    rq_wait_ft_sensor_steady(2000)
    zero_ftsensor()
    sleep(0.1)
    # end: URCap Program Node
    # begin: URCap Program Node
    #   Source: Robotiq_Copilot, 1.22.1.14215, Robotiq Inc.
    #   Type: Find Surface
    $ 80 "Find Surface"
    zero_ftsensor()
    sleep(0.1)
    surface_found = rq_linear_search_urcap("Z+", 10.000, 0.005000, 0.100000, 1)
    storevar.setvariablepose("rq_findSurface_ef5e6fd5-1d3d-43c2-9922-b9c2fd55821a_exitPosition", get_actual_tcp_pose())
    $ 81 "'Add Stop conditions from the Find Surface node'" "noBreak"
    # 'Add Stop conditions from the Find Surface node'
    # end: URCap Program Node
    # begin: URCap Program Node
    #   Source: Robotiq_Copilot, 1.22.1.14215, Robotiq Inc.
    #   Type: Finishing Tool Control
    $ 82 "Start tool"
    set_standard_digital_out(0, True)
    # end: URCap Program Node
    $ 83 "Wait: 0.5"
    sleep(0.5)
    $ 84 "Force"
    sleep(0.02)
    zero_ftsensor()
    force_mode(tool_pose(), [0, 0, 1, 0, 0, 0], [0.0, 0.0, 5.0, 0.0, 0.0, 0.0], 2, [0.1, 0.1, 0.15, 0.3490658503988659, 0.3490658503988659, 0.3490658503988659])
    $ 85 "Waypoint_7" "noBreak"
    set_tcp(p[0.00318,0.11464,0.09820000000000001,-0.7853981633974483,0.0,0.0])
    movel(pose_trans(CubeFront, pose_trans(p[-.005597006121, -.192408094989, .653246871754, -1.571622694982, -.002967386491, .002471774867], Waypoint_7_p)), a=1.2, v=0.05)
    end_force_mode()
    stopl(5.0)
    # begin: URCap Program Node
    #   Source: Robotiq_Copilot, 1.22.1.14215, Robotiq Inc.
    #   Type: Finishing Tool Control
    $ 86 "Stop tool"
    set_standard_digital_out(0, False)
    # end: URCap Program Node
    $ 87 "Waypoint_13" "breakAfter"
    set_tcp(p[0.00318,0.11464,0.09820000000000001,-0.7853981633974483,0.0,0.0])
    movel(pose_trans(CubeFront, pose_trans(p[-.002001169423, -.178123008725, .618090231485, -1.568699287997, .013964727372, .007428573496], Waypoint_13_p)), a=1.2, v=0.25)
    $ 88 "Waypoint_9" "breakAfter"
    set_tcp(p[0.00318,0.11464,0.09820000000000001,-0.7853981633974483,0.0,0.0])
    movel(pose_trans(CubeFront, pose_trans(p[-.002001169423, -.178123008725, .618090231485, -1.568699287997, .013964727372, .007428573496], Waypoint_9_p)), a=1.2, v=0.25)
    $ 89 "clear" "breakAfter"
    set_tcp(p[0.00318,0.11464,0.09820000000000001,-0.7853981633974483,0.0,0.0])
    movel(pose_trans(CubeFront, pose_trans(p[.002249871974, -.169402369556, .608081756259, .020435046430, 2.223511403835, 2.209446612627], clear_p)), a=1.2, v=0.25)
  end
  def SprayFront():
    $ 90 "SprayFront" "noBreak"
    $ 91 "SprayFront"
    $ 92 "MoveJ"
    $ 93 "clear" "breakAfter"
    set_tcp(p[0.00318,0.11464,0.09820000000000001,-0.7853981633974483,0.0,0.0])
    movej(get_inverse_kin(pose_trans(CubeFront, pose_trans(p[.002249871974, -.169402369556, .608081756259, .020435046430, 2.223511403835, 2.209446612627], clear_p)), qnear=clear_q), a=1.3962634015954636, v=1.0471975511965976)
    $ 94 "MoveJ"
    $ 95 "Waypoint_10" "breakAfter"
    set_tcp(p[0.020839023181949995,-0.027139950822234082,0.10599373590389219,0.12258870209179472,1.1769383890382668,2.869747076630172])
    movej(get_inverse_kin(pose_trans(CubeFront, pose_trans(p[-.002001169423, -.178123008725, .618090231485, -1.568699287997, .013964727372, .007428573496], Waypoint_10_p)), qnear=Waypoint_10_q), a=1.3962634015954636, v=1.0471975511965976)
    $ 96 "Set DO[1]=On"
    set_standard_digital_out(1, True)
    $ 97 "MoveL"
    $ 98 "Waypoint_12" "breakAfter"
    movel(pose_trans(CubeFront, pose_trans(p[-.002001169423, -.178123008725, .618090231485, -1.568699287997, .013964727372, .007428573496], Waypoint_12_p)), a=1.2, v=0.1)
    $ 99 "Set DO[1]=Off"
    set_standard_digital_out(1, False)
    $ 100 "MoveJ"
    $ 101 "Waypoint_21" "breakAfter"
    set_tcp(p[0.020839023181949995,-0.027139950822234082,0.10599373590389219,0.12258870209179472,1.1769383890382668,2.869747076630172])
    movej(get_inverse_kin(pose_trans(CubeFront, pose_trans(p[-.002001169423, -.178123008725, .618090231485, -1.568699287997, .013964727372, .007428573496], Waypoint_21_p)), qnear=Waypoint_21_q), a=1.3962634015954636, v=1.0471975511965976)
    $ 102 "Set DO[1]=On"
    set_standard_digital_out(1, True)
    $ 103 "MoveL"
    $ 104 "Waypoint_22" "breakAfter"
    set_tcp(p[0.020839023181949995,-0.027139950822234082,0.10599373590389219,0.12258870209179472,1.1769383890382668,2.869747076630172])
    movel(pose_trans(CubeFront, pose_trans(p[-.002001169423, -.178123008725, .618090231485, -1.568699287997, .013964727372, .007428573496], Waypoint_22_p)), a=1.2, v=0.1)
    $ 105 "Set DO[1]=Off"
    set_standard_digital_out(1, False)
    $ 106 "MoveJ"
    $ 107 "Waypoint_23" "breakAfter"
    set_tcp(p[0.020839023181949995,-0.027139950822234082,0.10599373590389219,0.12258870209179472,1.1769383890382668,2.869747076630172])
    movej(get_inverse_kin(pose_trans(CubeFront, pose_trans(p[-.002001169423, -.178123008725, .618090231485, -1.568699287997, .013964727372, .007428573496], Waypoint_23_p)), qnear=Waypoint_23_q), a=1.3962634015954636, v=1.0471975511965976)
    $ 108 "Set DO[1]=On"
    set_standard_digital_out(1, True)
    $ 109 "MoveL"
    $ 110 "Waypoint_24" "breakAfter"
    set_tcp(p[0.020839023181949995,-0.027139950822234082,0.10599373590389219,0.12258870209179472,1.1769383890382668,2.869747076630172])
    movel(pose_trans(CubeFront, pose_trans(p[-.002001169423, -.178123008725, .618090231485, -1.568699287997, .013964727372, .007428573496], Waypoint_24_p)), a=1.2, v=0.1)
    $ 111 "Set DO[1]=Off"
    set_standard_digital_out(1, False)
    $ 112 "MoveJ"
    $ 113 "clear" "breakAfter"
    movej(clear_q, a=1.3962634015954636, v=1.0471975511965976)
    $ 114 "MoveJ"
    $ 115 "Waypoint_26" "breakAfter"
    set_tcp(p[0.020839023181949995,-0.027139950822234082,0.10599373590389219,0.12258870209179472,1.1769383890382668,2.869747076630172])
    movej(get_inverse_kin(pose_trans(CubeFront, pose_trans(p[-.002001169423, -.178123008725, .618090231485, -1.568699287997, .013964727372, .007428573496], Waypoint_26_p)), qnear=Waypoint_26_q), a=1.3962634015954636, v=1.0471975511965976)
    $ 116 "Set DO[1]=On"
    set_standard_digital_out(1, True)
    $ 117 "MoveL"
    $ 118 "Waypoint_25" "breakAfter"
    set_tcp(p[0.020839023181949995,-0.027139950822234082,0.10599373590389219,0.12258870209179472,1.1769383890382668,2.869747076630172])
    movel(pose_trans(CubeFront, pose_trans(p[-.002001169423, -.178123008725, .618090231485, -1.568699287997, .013964727372, .007428573496], Waypoint_25_p)), a=1.2, v=0.1)
    $ 119 "Set DO[1]=Off"
    set_standard_digital_out(1, False)
    $ 120 "MoveJ"
    $ 121 "clear" "breakAfter"
    movej(clear_q, a=1.3962634015954636, v=1.0471975511965976)
  end
  def SprayRebate():
    $ 122 "SprayRebate" "noBreak"
    $ 123 "SprayRebate"
    $ 124 "MoveJ"
    $ 125 "clear" "breakAfter"
    movej(clear_q, a=1.3962634015954636, v=1.0471975511965976)
    $ 126 "MoveJ"
    $ 127 "Waypoint_28" "breakAfter"
    set_tcp(p[0.020839023181949995,-0.027139950822234082,0.10599373590389219,0.12258870209179472,1.1769383890382668,2.869747076630172])
    movej(get_inverse_kin(pose_trans(CubeFront, pose_trans(p[-.002001169423, -.178123008725, .618090231485, -1.568699287997, .013964727372, .007428573496], Waypoint_28_p)), qnear=Waypoint_28_q), a=1.3962634015954636, v=1.0471975511965976)
    $ 128 "Set DO[1]=On"
    set_standard_digital_out(1, True)
    $ 129 "MoveL"
    $ 130 "Waypoint_27" "breakAfter"
    set_tcp(p[0.020839023181949995,-0.027139950822234082,0.10599373590389219,0.12258870209179472,1.1769383890382668,2.869747076630172])
    movel(pose_trans(CubeFront, pose_trans(p[-.002001169423, -.178123008725, .618090231485, -1.568699287997, .013964727372, .007428573496], Waypoint_27_p)), a=1.2, v=0.1)
    $ 131 "Set DO[1]=Off"
    set_standard_digital_out(1, False)
    $ 132 "MoveJ"
    $ 133 "Waypoint_29" "breakAfter"
    set_tcp(p[0.020839023181949995,-0.027139950822234082,0.10599373590389219,0.12258870209179472,1.1769383890382668,2.869747076630172])
    movej(get_inverse_kin(pose_trans(CubeFront, pose_trans(p[-.002001169423, -.178123008725, .618090231485, -1.568699287997, .013964727372, .007428573496], Waypoint_29_p)), qnear=Waypoint_29_q), a=1.3962634015954636, v=1.0471975511965976)
    $ 134 "Set DO[1]=On"
    set_standard_digital_out(1, True)
    $ 135 "MoveL"
    $ 136 "Waypoint_30" "breakAfter"
    set_tcp(p[0.020839023181949995,-0.027139950822234082,0.10599373590389219,0.12258870209179472,1.1769383890382668,2.869747076630172])
    movel(pose_trans(CubeFront, pose_trans(p[-.002001169423, -.178123008725, .618090231485, -1.568699287997, .013964727372, .007428573496], Waypoint_30_p)), a=1.2, v=0.1)
    $ 137 "Set DO[1]=Off"
    set_standard_digital_out(1, False)
    $ 138 "MoveJ"
    $ 139 "clear" "breakAfter"
    movej(clear_q, a=1.3962634015954636, v=1.0471975511965976)
    $ 140 "MoveJ"
    $ 141 "Waypoint_32" "breakAfter"
    set_tcp(p[0.020839023181949995,-0.027139950822234082,0.10599373590389219,0.12258870209179472,1.1769383890382668,2.869747076630172])
    movej(get_inverse_kin(pose_trans(CubeFront, pose_trans(p[-.002001169423, -.178123008725, .618090231485, -1.568699287997, .013964727372, .007428573496], Waypoint_32_p)), qnear=Waypoint_32_q), a=1.3962634015954636, v=1.0471975511965976)
    $ 142 "Set DO[1]=On"
    set_standard_digital_out(1, True)
    $ 143 "MoveL"
    $ 144 "Waypoint_33" "breakAfter"
    set_tcp(p[0.020839023181949995,-0.027139950822234082,0.10599373590389219,0.12258870209179472,1.1769383890382668,2.869747076630172])
    movel(pose_trans(CubeFront, pose_trans(p[-.002001169423, -.178123008725, .618090231485, -1.568699287997, .013964727372, .007428573496], Waypoint_33_p)), a=1.2, v=0.1)
    $ 145 "Set DO[1]=Off"
    set_standard_digital_out(1, False)
    $ 146 "MoveJ"
    $ 147 "clear" "breakAfter"
    movej(clear_q, a=1.3962634015954636, v=1.0471975511965976)
  end
  def SandFront():
    $ 148 "SandFront" "noBreak"
    $ 149 "sandFront"
    $ 150 "MoveJ"
    $ 151 "clear" "breakAfter"
    set_tcp(p[0.00318,0.11464,0.09820000000000001,-0.7853981633974483,0.0,0.0])
    movej(get_inverse_kin(pose_trans(CubeFront, pose_trans(p[.002249871974, -.169402369556, .608081756259, .020435046430, 2.223511403835, 2.209446612627], clear_p)), qnear=clear_q), a=1.3962634015954636, v=1.0471975511965976)
    $ 152 "MoveL"
    $ 153 "Waypoint_1" "breakAfter"
    set_tcp(p[0.00318,0.11464,0.09820000000000001,-0.7853981633974483,0.0,0.0])
    movel(pose_trans(CubeFront, pose_trans(p[-.005597006121, -.192408094989, .653246871754, -1.571622694982, -.002967386491, .002471774867], Waypoint_1_p)), a=1.2, v=0.25)
    # begin: URCap Program Node
    #   Source: Robotiq_Copilot, 1.22.1.14215, Robotiq Inc.
    #   Type: Zero FT Sensor
    $ 154 "Zero FT Sensor"

    rq_wait_ft_sensor_steady(2000)
    zero_ftsensor()
    sleep(0.1)
    # end: URCap Program Node
    # begin: URCap Program Node
    #   Source: Robotiq_Copilot, 1.22.1.14215, Robotiq Inc.
    #   Type: Find Surface
    $ 155 "Find Surface"
    surface_found = rq_linear_search_urcap("Z+", 10.000, 0.005000, 0.100000, 1)
    storevar.setvariablepose("rq_findSurface_7eeff1a3-6c12-4ed4-8857-ddcfb00799c6_exitPosition", get_actual_tcp_pose())
    $ 156 "'Add Stop conditions from the Find Surface node'" "noBreak"
    # 'Add Stop conditions from the Find Surface node'
    # end: URCap Program Node
    # begin: URCap Program Node
    #   Source: Robotiq_Copilot, 1.22.1.14215, Robotiq Inc.
    #   Type: Finishing Tool Control
    $ 157 "Start tool"
    set_standard_digital_out(0, True)
    # end: URCap Program Node
    $ 158 "Wait: 0.5"
    sleep(0.5)
    $ 159 "MoveL"
    $ 160 "Force"
    sleep(0.02)
    zero_ftsensor()
    force_mode(tool_pose(), [0, 0, 1, 0, 0, 0], [0.0, 0.0, 5.0, 0.0, 0.0, 0.0], 2, [0.1, 0.1, 0.15, 0.3490658503988659, 0.3490658503988659, 0.3490658503988659])
    $ 161 "Waypoint_34" "noBreak"
    set_tcp(p[0.00318,0.11464,0.09820000000000001,-0.7853981633974483,0.0,0.0])
    movel(pose_trans(CubeFront, pose_trans(p[.002249871974, -.169402369556, .608081756259, .020435046430, 2.223511403835, 2.209446612627], Waypoint_34_p)), a=1.2, v=0.06)
    $ 162 "Waypoint_37" "noBreak"
    set_tcp(p[0.00318,0.11464,0.09820000000000001,-0.7853981633974483,0.0,0.0])
    movel(pose_trans(CubeFront, pose_trans(p[.002249871974, -.169402369556, .608081756259, .020435046430, 2.223511403835, 2.209446612627], Waypoint_37_p)), a=1.2, v=0.06)
    $ 163 "Waypoint_36" "noBreak"
    set_tcp(p[0.00318,0.11464,0.09820000000000001,-0.7853981633974483,0.0,0.0])
    movel(pose_trans(CubeFront, pose_trans(p[.002249871974, -.169402369556, .608081756259, .020435046430, 2.223511403835, 2.209446612627], Waypoint_36_p)), a=1.2, v=0.06)
    $ 164 "Waypoint_1" "noBreak"
    set_tcp(p[0.00318,0.11464,0.09820000000000001,-0.7853981633974483,0.0,0.0])
    movel(pose_trans(CubeFront, pose_trans(p[-.005597006121, -.192408094989, .653246871754, -1.571622694982, -.002967386491, .002471774867], Waypoint_1_p)), a=1.2, v=0.06)
    # begin: URCap Program Node
    #   Source: Robotiq_Copilot, 1.22.1.14215, Robotiq Inc.
    #   Type: Finishing Tool Control
    $ 165 "Stop tool" "noBreak"
    set_standard_digital_out(0, False)
    # end: URCap Program Node
    end_force_mode()
    stopl(5.0)
    $ 166 "Direction: Tool Z-"
    global move_thread_flag_166=0
    thread move_thread_166():
      enter_critical
      move_thread_flag_166 = 1
      local towardsPos=calculate_point_to_move_towards(get_forward_kin(), [0.0,0.0,-1.0], 0.025)
      movel(towardsPos, a=1.2, v=0.06)
      move_thread_flag_166 = 2
      exit_critical
    end
    move_thread_flag_166 = 0
    move_thread_han_166 = run move_thread_166()
    while (True):
      sleep(1.0E-10)
      if (move_thread_flag_166 > 1):
        join move_thread_han_166
        $ 167 "Until (distance)"
        break
      end
      sync()
    end
    $ 168 "MoveJ"
    $ 169 "clear" "breakAfter"
    movej(get_inverse_kin(pose_trans(CubeFront, pose_trans(p[.002249871974, -.169402369556, .608081756259, .020435046430, 2.223511403835, 2.209446612627], clear_p)), qnear=clear_q), a=1.3962634015954636, v=1.0471975511965976)
  end
  def StartSpray():
    $ 170 "StartSpray" "noBreak"
    $ 171 "Set DO[1]=On"
    set_standard_digital_out(1, True)
    $ 172 "Wait: 0.3"
    sleep(0.3)
  end
  def stopSpray():
    $ 173 "stopSpray" "noBreak"
    $ 174 "Set DO[1]=Off"
    set_standard_digital_out(1, False)
    $ 175 "Wait: 0.3"
    sleep(0.3)
  end
  thread EventThread():
    while (True):
      if (get_standard_digital_in(1) !=   True  ):
        $ 45 "Set DO[0]=Off"
        set_standard_digital_out(0, False)
        $ 46 "Set DO[1]=Off"
        set_standard_digital_out(1, False)
        $ 47 "Halt"
        halt
      end
      sync()
    end
  end
  eventThread = run EventThread()
  while (True):
    $ 1 "Robot Program"
    $ 2 "Main"
    $ 3 "MoveJ"
    $ 4 "clear" "breakAfter"
    set_tcp(p[0.00318,0.11464,0.09820000000000001,-0.7853981633974483,0.0,0.0])
    movej(get_inverse_kin(pose_trans(CubeFront, pose_trans(p[.002249871974, -.169402369556, .608081756259, .020435046430, 2.223511403835, 2.209446612627], clear_p)), qnear=clear_q), a=1.3962634015954636, v=1.0471975511965976)
    # begin: URCap Program Node
    #   Source: Robotiq_Copilot, 1.22.1.14215, Robotiq Inc.
    #   Type: Zero FT Sensor
    $ 5 "Zero FT Sensor"

    rq_wait_ft_sensor_steady(2000)
    zero_ftsensor()
    sleep(0.1)
    # end: URCap Program Node
    $ 6 "CubeFront≔CubeFront"
    global CubeFront=CubeFront
    $ 7 "Call SandFront"
    SandFront()
    $ 8 "CubeFront≔SandBack"
    global CubeFront=SandBack
    $ 9 "Call SandFront"
    SandFront()
  end
end
